{attribute 'qualified_only'}
TYPE E_IPM_States :
(
    Unknown := 0,
    OUT := 1,
    TARGET1 := 2,
    TARGET2 := 3,
    TARGET3 := 4,
    TARGET4 := 5
) UINT;
END_TYPE

(* stored: Version 1.1.0.1
   DUT E_IPM_States: Id {30889ac4-43ab-4289-9f65-9c3e86895012} *)
